PROGRAM MAIN
VAR
	//Client
	//fbhttpClient : FB_IotHttpClient := (sHostName:='postman-echo.com',
	//							  	bKeepAlive:=TRUE, tConnectionTimeout:=T#10S);
									
	//Eton
	fbhttpClient : FB_IotHttpClient := (sHostName:='api.em.eaton.com',
								  	bKeepAlive:=TRUE, tConnectionTimeout:=T#10S);		
				
	//Get Request
	fbRequest : FB_IotHttpRequest;		
	state : (IDLE, SEND_REQUEST, WAIT_FOR_RESPONSE, READ_RESPONSE,ERROR,FORMATER);			
	sendGetRequest: BOOL;
	debugContent : STRING(511);
	fbJsonParser : FB_JsonDomParser;
	jsonDoc				: SJsonValue;
	jsonArgsMember				: SJsonValue;
	jsonFoo2 : SJsonValue;
	results : STRING;
	
	//JSON Formater
	fbJsonWriter         : FB_JsonSaxWriter;
	sendData                : STRING(2000);
	
END_VAR

//PostmanEco();
MockServer();
//EtonSmartBreaker();

END_PROGRAM

(* stored: Version 1.1.0.1, ProductVersion 3.1.4024.12
   POU MAIN: Id {3d5404ea-3a8c-486d-8750-2451566905c2}, SpecialFunc None *)
